(* IEC 61131-3 sources: Caravan/Archiv/12-04-19/Stations/MachineControl/MachineControl/Class/HmiVarList35, 1 file *)

(* ---- HmiVarList35.st ---- *)
(*!
<Class
	Name               = "HmiVarList35"
	Revision           = "0.4"
	RealtimeTask       = "false"
	CyclicTask         = "false"
	BackgroundTask     = "false"
	Sigmatek           = "true"
	OSInterface        = "false"
	HighPriority       = "false"
	Automatic          = "false"
	UpdateMode         = "Prescan"
	SharedCommandTable = "true"
	Objectsize         = "(284,120)">
	<Channels>
		<Server Name="ByteSize" Visualized="false" Initialize="false" WriteProtected="true" Retentive="false"/>
		<Server Name="ClassSvr" Visualized="false" Initialize="false" WriteProtected="true" Retentive="false"/>
	</Channels>
	<RevDoku>
		<Owner Company="sigmatek" Author="kolott"/>
		<Dokumentation Revision="0.4" Date="2017-11-28" Author="kolott" Company="sigmatek" Description="inc of ClassSvr during add of variables"/>
		<Dokumentation Revision="0.3" Date="2014-08-07" Author="kolott" Company="sigmatek" Description="server of type ENUM will work as well"/>
		<Dokumentation Revision="0.2" Date="2014-03-28" Author="kolott" Company="sigmatek" Description="server ByteSize added"/>
		<Dokumentation Revision="0.1" Date="2014-03-26" Author="kolott" Company="sigmatek" Description="innovation: ClassSvr will represent number of used servers in HMI"/>
	</RevDoku>
</Class>
*)
HmiVarList35 : CLASS
  //Servers:
	ClassSvr 	: SvrChCmd_DINT;
	ByteSize 	: SvrCh_UDINT;
  //Clients:
  //Variables:
		Ptr 	: ^void;
		xData : ARRAY [0..20000] OF USINT;

  //Functions:

	FUNCTION GLOBAL Free;

	FUNCTION GLOBAL Start;

	FUNCTION GLOBAL AddEntry
		VAR_INPUT
			og 	: DINT;
			ug 	: DINT;
			textdescribing 	: UINT;
			textunit 	: UINT;
		END_VAR
		VAR_OUTPUT
			retcode 	: UDINT;
		END_VAR;

	FUNCTION GLOBAL End
		VAR_OUTPUT
			retcode 	: ^void;
		END_VAR;
  //Tables:
	FUNCTION @STD
		VAR_OUTPUT
			ret_code	: CONFSTATES;
		END_VAR;
	FUNCTION GLOBAL TAB @CT_;
END_CLASS;

#includeC "..\LseEasy\Create.h"

#define MAXVARNUMBER35  ((sizeof(xData) - sizeof(_BOX_VARLIST)) / sizeof(_BOX_VARLIST_ENTRY)) //1024

FUNCTION GLOBAL HmiVarList35::Free

  Start();

END_FUNCTION

FUNCTION GLOBAL HmiVarList35::Start

  Ptr      := NIL;
  ClassSvr := 0;
  ByteSize := 0;

END_FUNCTION

FUNCTION GLOBAL HmiVarList35::AddEntry
	VAR_INPUT
		og 	: DINT;
		ug 	: DINT;
		textdescribing 	: UINT;
		textunit 	: UINT;
	END_VAR
	VAR_OUTPUT
		retcode 	: UDINT;
	END_VAR
  var
    pvar : ^_BOX_VARLIST;
    pdst : ^_BOX_VARLIST_ENTRY;
  end_var

  retcode := 16#FFFFFFFF;

  if(Ptr = NIL) then
    Ptr := #xData[0];
    _memset(Ptr, 0, sizeof(xData));
    pvar$^void := Ptr;
    pvar^.no           := 0;
    pvar^.boxhdr.size  := 0;
    pvar^.boxhdr.crc32 := 0;
  end_if;

  pvar$^void := Ptr;
  if(pvar^.no < MAXVARNUMBER35) then
    pdst     := #pvar^.data[0]; // decieve boundexceed
    pdst     += pvar^.no * sizeof(_BOX_VARLIST_ENTRY);
    pdst^.og := og;
    pdst^.ug := ug;
    pdst^.textdescribing := textdescribing;
    pdst^.textunit       := textunit;
    retcode := pvar^.no;
    pvar^.no += 1;
    ClassSvr += 1;
  end_if;

END_FUNCTION

FUNCTION GLOBAL HmiVarList35::End
	VAR_OUTPUT
		retcode 	: ^void;
	END_VAR
  var
    pvar : ^_BOX_VARLIST;
  end_var

  if(Ptr <> NIL) then
    pvar$^void := Ptr;
    ClassSvr   := pvar^.no;
    pvar^.boxhdr.size := 0;
    end_BIGBOX_HEADER(#pvar^.boxhdr, sizeof(_BOX_VARLIST) - sizeof(pvar^.data) + (pvar^.no * sizeof(_BOX_VARLIST_ENTRY)));
    ByteSize := pvar^.boxhdr.size;
  end_if;

  retcode := Ptr;

END_FUNCTION
